PROGRAM P30_ManualControl
VAR_INPUT
	state_Control	: INT; // 10:EnableControl
END_VAR
VAR
	i 	: INT;
END_VAR

//FOR i:=1 TO 26 DO
//	IF GVL_IO.aMaxValueController[i] <> 0 THEN
//		GVL_IO.aAnalogOutputIO[i] := LREAL_TO_INT(GVL_IO.aController[i].rControlValue); //Write to Device
		
//		GVL_IO.aController_PV[i] := (GVL_IO.aAnalogInputIO[i] / GVL_IO.KL3464MaxValueH) * GVL_IO.aMaxValueController[i]);
//		GVL_IO.aController_CV[i] := LREAL_TO_REAL((GVL_IO.aController[i].rControlValue / GVL_IO.KL3464MaxValueH)*GVL_IO.aMaxValueController[i]);
//		GVL_IO.aController[i]();
//	END_IF
//END_FOR

//(* Reactor Susceptor Temperature *)
//IF ( GVL_IO.aController_CV[27] > 10 ) THEN
//	GVL_IO.aDigitalOutputIO[2].0 := TRUE;
//ELSE
//	GVL_IO.aDigitalOutputIO[2].0 := FALSE;
//END_IF

//GVL_IO.wE3508_CV := LREAL_TO_WORD(GVL_IO.aController[27].rControlValue); //Write to Temperature Controller

//GVL_IO.aController_PV[27] := WORD_TO_REAL(GVL_IO.wE3508_PV);
//GVL_IO.aController_CV[27] := WORD_TO_REAL(GVL_IO.wE3508_CV);
//GVL_IO.aController[27]();
				
//(* Reactor Pressure Control *)
//GVL_IO.wIqPlus_CV := LREAL_TO_WORD(GVL_IO.aController[28].rControlValue); //Write to Pressure Controller

//GVL_IO.aController_PV[28] := WORD_TO_REAL(GVL_IO.wIqPlus_CDG2_PV);
//GVL_IO.aController_CV[28] := WORD_TO_REAL(GVL_IO.wIqPlus_CV);
//GVL_IO.aController[28]();

//(* Suceptor Rotation Control *)				
//GVL_IO.rRotation_ControlValue := LREAL_TO_REAL(GVL_IO.aController[29].rControlValue); //Write to Rotation Controller (rpm)

//GVL_IO.aController_PV[29] := GVL_IO.nRotation_Converted_PV;
//GVL_IO.aController_CV[29] := GVL_IO.rRotation_ControlValue;
//GVL_IO.aController[29]();

END_PROGRAM

(* stored: Version 1.1.0.1, ProductVersion 3.1.4024.15
   POU P30_ManualControl: Id {98ee4f4f-99e9-426e-9dfa-55ddf51d552b}, SpecialFunc None *)
